FUNCTION_BLOCK UT_AuxiliaryInputMapping_Type_09_CombinedAnalog_Ret50perc (* Type 9 CombinedAnalog_Ret50perc Two way analog - return to centre position - with latching *)
  (* Standard: ISO 11783-6; Classification: AUX – ISO 11783-6; Function: All Inputs; Type: UT according to ISO 11783-6; Description: - Type 9 CombinedAnalog_Ret50perc Two way analog - return to centre position - with latching Applicable AUX-N only * maps to IW IW - Input WORD (16 Bit) * Maps to IX *)
  (* Version 1.0, 2018-12-05, Jose Cabral *)
  (* Version 1.1, 2022-08-04, Franz Höpfinger, HR Agrartechnik GmbH *)
  (* Version 1.2, 2023-01-05, Franz Höpfinger, HR Agrartechnik GmbH *)
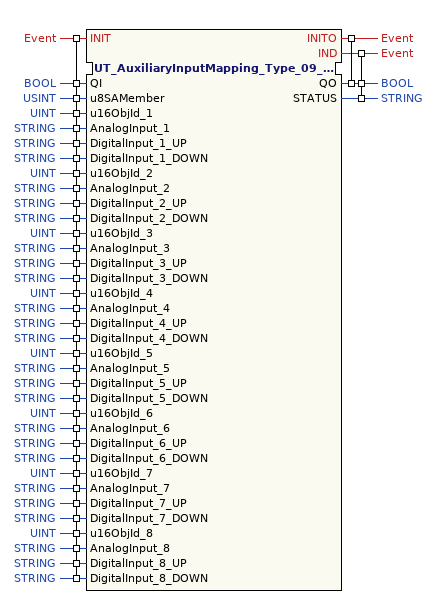
  EVENT_INPUT
    INIT WITH QI, u8SAMember, u16ObjId_1, AnalogInput_1, DigitalInput_1_UP, DigitalInput_1_DOWN, u16ObjId_2, AnalogInput_2, DigitalInput_2_UP, DigitalInput_2_DOWN, u16ObjId_3, AnalogInput_3, DigitalInput_3_UP, DigitalInput_3_DOWN, u16ObjId_4, AnalogInput_4, DigitalInput_4_UP, DigitalInput_4_DOWN, u16ObjId_5, AnalogInput_5, DigitalInput_5_UP, DigitalInput_5_DOWN, u16ObjId_6, AnalogInput_6, DigitalInput_6_UP, DigitalInput_6_DOWN, u16ObjId_7, AnalogInput_7, DigitalInput_7_UP, DigitalInput_7_DOWN, u16ObjId_8, AnalogInput_8, DigitalInput_8_UP, DigitalInput_8_DOWN; (* Service Initialization *)
  END_EVENT
  EVENT_OUTPUT
    INITO WITH QO; (* Initialization Confirm *)
    IND WITH QO, STATUS; (* Indication from Resource *)
  END_EVENT
  VAR_INPUT
    QI : BOOL; (* Event Input Qualifier *)
    u8SAMember : USINT := 255; (* Dummy !, set to 255 if in doubt. 0 deactivates FB. *)
    u16ObjId_1 : UINT; (* Object ID of Input 1 *)
    AnalogInput_1 : STRING; (* Identifier for Input 1 *)
    DigitalInput_1_UP : STRING; (* Identifier for Input 1 UP *)
    DigitalInput_1_DOWN : STRING; (* Identifier for Input 1 DOWN *)
    u16ObjId_2 : UINT; (* Object ID of Input 2 *)
    AnalogInput_2 : STRING; (* Identifier for Input 2 *)
    DigitalInput_2_UP : STRING; (* Identifier for Input 2 UP *)
    DigitalInput_2_DOWN : STRING; (* Identifier for Input 2 DOWN *)
    u16ObjId_3 : UINT; (* Object ID of Input 3 *)
    AnalogInput_3 : STRING; (* Identifier for Input 3 *)
    DigitalInput_3_UP : STRING; (* Identifier for Input 3 UP *)
    DigitalInput_3_DOWN : STRING; (* Identifier for Input 3 DOWN *)
    u16ObjId_4 : UINT; (* Object ID of Input 4 *)
    AnalogInput_4 : STRING; (* Identifier for Input 4 *)
    DigitalInput_4_UP : STRING; (* Identifier for Input 4 UP *)
    DigitalInput_4_DOWN : STRING; (* Identifier for Input 4 DOWN *)
    u16ObjId_5 : UINT; (* Object ID of Input 5 *)
    AnalogInput_5 : STRING; (* Identifier for Input 5 *)
    DigitalInput_5_UP : STRING; (* Identifier for Input 5 UP *)
    DigitalInput_5_DOWN : STRING; (* Identifier for Input 5 DOWN *)
    u16ObjId_6 : UINT; (* Object ID of Input 6 *)
    AnalogInput_6 : STRING; (* Identifier for Input 6 *)
    DigitalInput_6_UP : STRING; (* Identifier for Input 6 UP *)
    DigitalInput_6_DOWN : STRING; (* Identifier for Input 6 DOWN *)
    u16ObjId_7 : UINT; (* Object ID of Input 7 *)
    AnalogInput_7 : STRING; (* Identifier for Input 7 *)
    DigitalInput_7_UP : STRING; (* Identifier for Input 7 UP *)
    DigitalInput_7_DOWN : STRING; (* Identifier for Input 7 DOWN *)
    u16ObjId_8 : UINT; (* Object ID of Input 8 *)
    AnalogInput_8 : STRING; (* Identifier for Input 8 *)
    DigitalInput_8_UP : STRING; (* Identifier for Input 8 UP *)
    DigitalInput_8_DOWN : STRING; (* Identifier for Input 8 DOWN *)
  END_VAR
  VAR_OUTPUT
    QO : BOOL; (* Event Output Qualifier *)
    STATUS : STRING; (* Service Status *)
  END_VAR
END_FUNCTION_BLOCK
